(* PLC project Tc3_EventLogger.F_GetEventClassName Demo, tc3-libraries-kb TwinCAT 3.1 *)
(* stored: creationDateTime 2026-05-11T01:00:00, modificationDateTime 2026-05-11T01:00:00 *)

PROGRAM P_Demo_F_GetEventClassName
  VAR
    fbF_GetEventClassName : F_GetEventClassName;  (* Tc3_EventLogger.F_GetEventClassName 实例 *)
    arg_nLangId : DINT;  (* VAR_INPUT nLangId *)
    arg_fbEventBase : REFERENCE TO FB_TcEventBase;  (* VAR_INPUT fbEventBase *)
    io_fbResult : FB_AsyncStrResult;  (* VAR_IN_OUT fbResult *)
  END_VAR

            // ============================================================
// Tc3_EventLogger.F_GetEventClassName 演示程序（FB 实例）
// ============================================================
// 验证步骤：
//   1. 引用 Tc3_EventLogger（及依赖类型所在库 Tc2_System 等）
//   2. 编译 + 登录
//   3. 按 doc.md 给 arg_* 赋值
//   4. 在线监视 out_* / io_* 输出
// ============================================================

fbF_GetEventClassName(
    nLangId := arg_nLangId,
    fbEventBase := arg_fbEventBase,
    fbResult := io_fbResult
);

          
END_PROGRAM
